PROGRAM MAIN
VAR
	outHard AT%Q* 		: INT := 0;
	outSoft				: INT := 0;
	inHard	AT%I*		: INT := 0;
	collision				: USINT := 0;
END_VAR

END_PROGRAM

(* stored: Version 1.1.0.1, ProductVersion 3.1.4024.11
   POU MAIN: Id {44f6d904-02dc-4765-8373-d446baf7443b}, SpecialFunc None *)
